% RSLogix 500 project SensorCalibration.RSS, saved by version 8.30.00.16 %
PROJECT "UNTITLED"    % processor: Bul.1763 MicroLogix 1100 Series B %

PROGRAM FILES
  LAD 2 "MAIN"  3 rungs
  LAD 4 "D OUT"  3 rungs
  LAD 5 "CONTROL"  12 rungs

DATA FILES
  O0 OUTPUT  4 elements
  I1 INPUT  6 elements
  S2 STATUS  66 elements
  B3 BINARY  1 elements
  T4 TIMER  2 elements
  C5 COUNTER  1 elements
  R6 CONTROL  1 elements
  N7 INTEGER  7 elements
  F8 FLOAT  2 elements

LADDER 2 "MAIN"
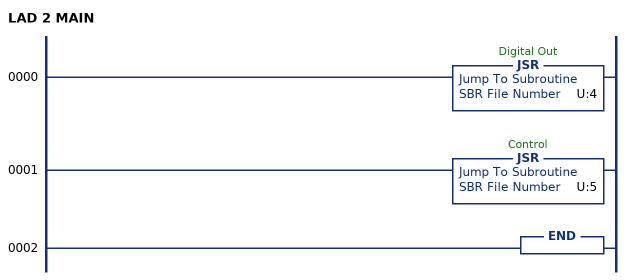
% Rung: 0 %
SOR JSR U:4 EOR
%   U:4  "Digital Out" %
% Rung: 1 %
SOR JSR U:5 EOR
%   U:5  "Control" %
% Rung: 2 %
SOR END EOR

LADDER 4 "D OUT"
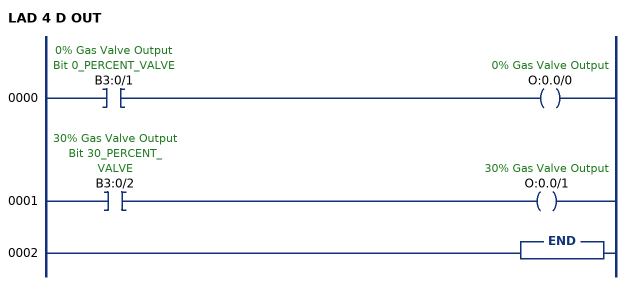
% Rung: 0 %
SOR XIC B3:0/1 OTE O:0.0/0 EOR
%   B3:0/1  0_PERCENT_VALVE  "0% Gas Valve Output Bit" %
%   O:0.0/0  "0% Gas Valve Output" %
% Rung: 1 %
SOR XIC B3:0/2 OTE O:0.0/1 EOR
%   B3:0/2  30_PERCENT_VALVE  "30% Gas Valve Output Bit" %
%   O:0.0/1  "30% Gas Valve Output" %
% Rung: 2 %
SOR END EOR

LADDER 5 "CONTROL"
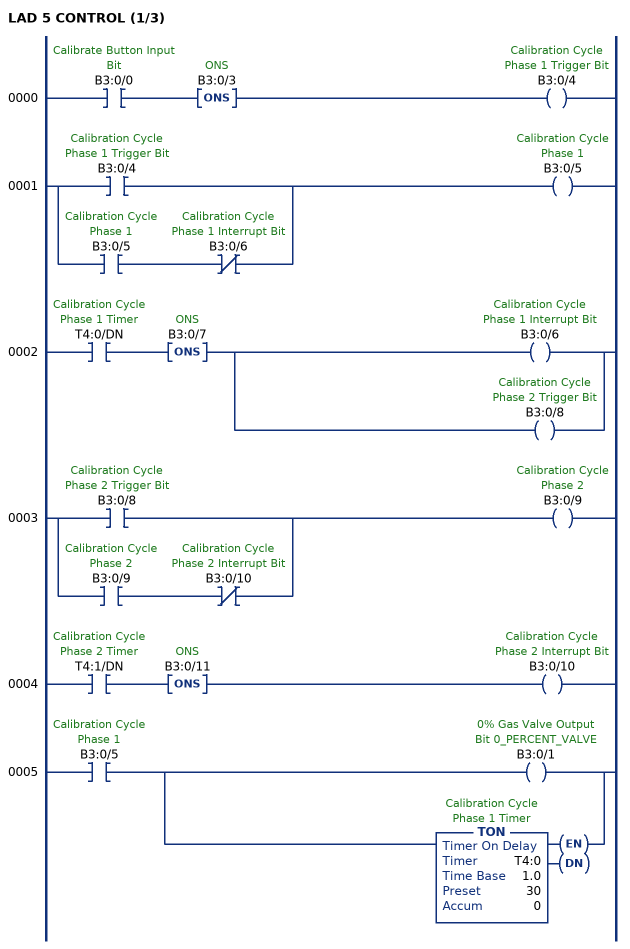
% Rung: 0 %
SOR XIC B3:0/0 ONS B3:0/3 OTE B3:0/4 EOR
%   B3:0/0  "Calibrate Button Input Bit" %
%   B3:0/3  "ONS" %
%   B3:0/4  "Calibration Cycle Phase 1 Trigger Bit" %
% Rung: 1 %
SOR BST XIC B3:0/4 NXB XIC B3:0/5 XIO B3:0/6 BND OTE B3:0/5 EOR
%   B3:0/4  "Calibration Cycle Phase 1 Trigger Bit" %
%   B3:0/5  "Calibration Cycle Phase 1" %
%   B3:0/6  "Calibration Cycle Phase 1 Interrupt Bit" %
% Rung: 2 %
SOR XIC T4:0/DN ONS B3:0/7 BST OTE B3:0/6 NXB OTE B3:0/8 BND EOR
%   T4:0  "Calibration Cycle Phase 1 Timer" %
%   B3:0/7  "ONS" %
%   B3:0/6  "Calibration Cycle Phase 1 Interrupt Bit" %
%   B3:0/8  "Calibration Cycle Phase 2 Trigger Bit" %
% Rung: 3 %
SOR BST XIC B3:0/8 NXB XIC B3:0/9 XIO B3:0/10 BND OTE B3:0/9 EOR
%   B3:0/8  "Calibration Cycle Phase 2 Trigger Bit" %
%   B3:0/9  "Calibration Cycle Phase 2" %
%   B3:0/10  "Calibration Cycle Phase 2 Interrupt Bit" %
% Rung: 4 %
SOR XIC T4:1/DN ONS B3:0/11 OTE B3:0/10 EOR
%   T4:1  "Calibration Cycle Phase 2 Timer" %
%   B3:0/11  "ONS" %
%   B3:0/10  "Calibration Cycle Phase 2 Interrupt Bit" %
% Rung: 5 %
SOR XIC B3:0/5 BST OTE B3:0/1 NXB TON T4:0 1.0 30 0 BND EOR
%   B3:0/5  "Calibration Cycle Phase 1" %
%   B3:0/1  0_PERCENT_VALVE  "0% Gas Valve Output Bit" %
%   T4:0  "Calibration Cycle Phase 1 Timer" %

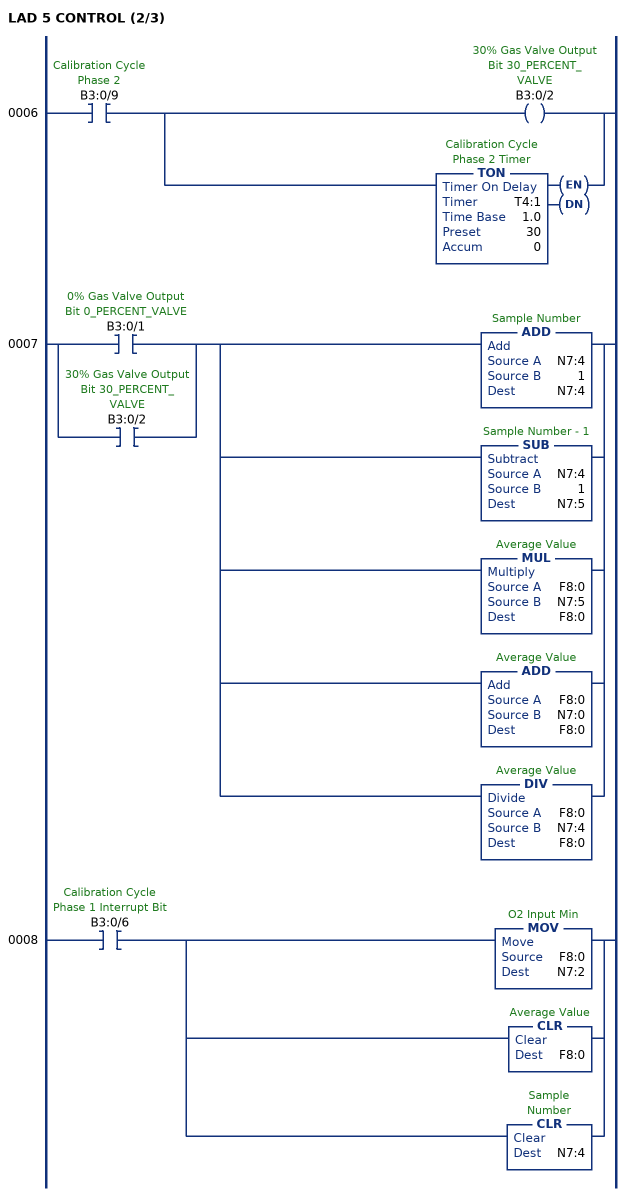
% Rung: 6 %
SOR XIC B3:0/9 BST OTE B3:0/2 NXB TON T4:1 1.0 30 0 BND EOR
%   B3:0/9  "Calibration Cycle Phase 2" %
%   B3:0/2  30_PERCENT_VALVE  "30% Gas Valve Output Bit" %
%   T4:1  "Calibration Cycle Phase 2 Timer" %
% Rung: 7 %
SOR BST XIC B3:0/1 NXB XIC B3:0/2 BND BST ADD N7:4 1 N7:4 NXB SUB N7:4 1 N7:5 NXB MUL F8:0 N7:5 F8:0 NXB ADD F8:0 N7:0 F8:0 NXB DIV F8:0 N7:4 F8:0 BND EOR
%   B3:0/1  0_PERCENT_VALVE  "0% Gas Valve Output Bit" %
%   B3:0/2  30_PERCENT_VALVE  "30% Gas Valve Output Bit" %
%   N7:4  "Sample Number" %
%   N7:5  "Sample Number - 1" %
%   F8:0  "Average Value" %
%   N7:0  "O2 Sensor Input Signal" %
% Rung: 8 %
SOR XIC B3:0/6 BST MOV F8:0 N7:2 NXB CLR F8:0 NXB CLR N7:4 BND EOR
%   B3:0/6  "Calibration Cycle Phase 1 Interrupt Bit" %
%   F8:0  "Average Value" %
%   N7:2  "O2 Input Min" %
%   N7:4  "Sample Number" %

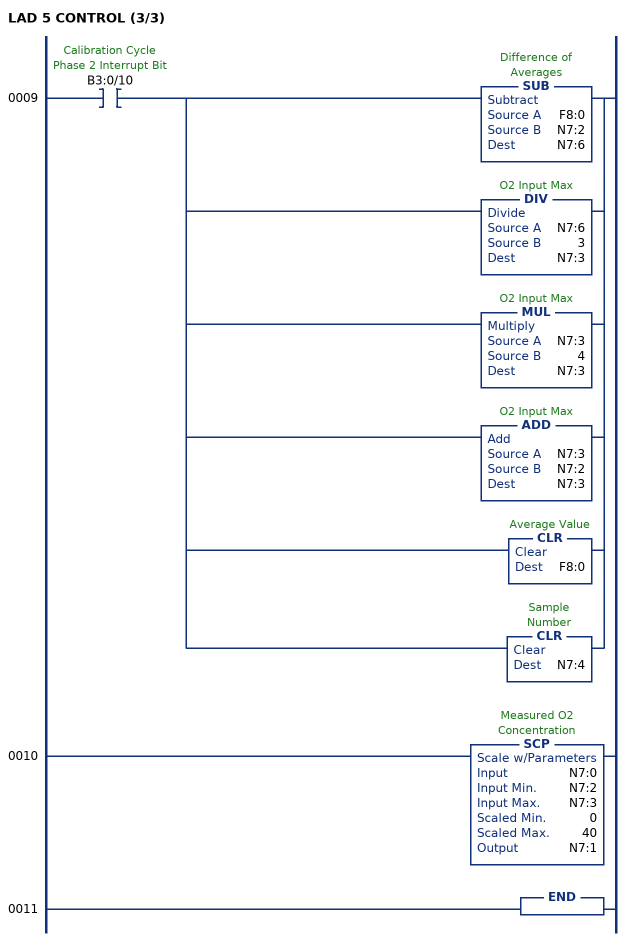
% Rung: 9 %
SOR XIC B3:0/10 BST SUB F8:0 N7:2 N7:6 NXB DIV N7:6 3 N7:3 NXB MUL N7:3 4 N7:3 NXB ADD N7:3 N7:2 N7:3 NXB CLR F8:0 NXB CLR N7:4 BND EOR
%   B3:0/10  "Calibration Cycle Phase 2 Interrupt Bit" %
%   F8:0  "Average Value" %
%   N7:2  "O2 Input Min" %
%   N7:6  "Difference of Averages" %
%   N7:3  "O2 Input Max" %
%   N7:4  "Sample Number" %
% Rung: 10 %
SOR SCP N7:0 N7:2 N7:3 0 40 N7:1 EOR
%   N7:0  "O2 Sensor Input Signal" %
%   N7:2  "O2 Input Min" %
%   N7:3  "O2 Input Max" %
%   N7:1  "Measured O2 Concentration" %
% Rung: 11 %
SOR END EOR

OTHER DOCUMENTED ADDRESSES
  F8:1  "4/3"

DATA TABLE (non-zero values as saved)
DATA T4
% .PRE .ACC %
% T4:0 % 30 0
% T4:1 % 30 0
DATA N7
% N7:0 % 8192 0 0 16383 0 0 0
